(* IEC 61131-3 sources: Lua/ (part 2) *)

(* ---- ValveControl.st ---- *)
REGION 预处理
    #"FP-valve-Product"(CLK := #"Comm-Valve"."bnt-run");
    #"FP-valve-Manual"(CLK := #"Comm-Valve"."bnt-stop");
    #"Valve-Timer"[0](IN := #"Comm-Valve".busy,PT := #"Screen-Time"."PT-pretime-v");
    #"Valve-Timer"[1](IN := #"Comm-Valve"."in-timer".%X1,PT := #"Screen-Time"."PT-opentime");
    #"Valve-Timer"[2](IN := #"Comm-Valve"."in-timer".%X2,PT := #"Screen-Time"."PT-delaytime");
    #"Valve-Timer"[3](IN := #"Comm-Valve"."in-timer".%X3,PT := #"Screen-Time"."PT-looptime");
    //阀组生产模式
    IF "Debug".Unit_estop_state[2] THEN
        IF (#"FP-valve-Product".Q OR #"Comm-run".todo) AND NOT #"Comm-Valve".busy THEN
            #"Comm-Valve".todo := 1;
        END_IF;
        IF #"Comm-Valve".todo THEN
            #"Comm-Valve".busy := 1;
            #"Comm-Valve".step := 1;
            #"Comm-Valve".todo := 0;
        END_IF;
    ELSE
        #"Comm-Valve"."in-timer" := 0;
        #"Comm-Valve".todo := 0;
        #"Comm-Valve".busy := 0;
        #"Comm-Valve".step := 0;
    END_IF;
    //阀组手动模式
    IF "Debug".Unit_estop_state[2] THEN
        IF (#"FP-valve-Manual".Q OR #"Comm-stop".todo) THEN
            #"Comm-Valve"."in-timer" := 0;
            #"Comm-Valve".todo := 0;
            #"Comm-Valve".busy := 0;
            #"Comm-Valve".step := 0;
            "V5002-O" := 0;
            "V5003-O" := 0;
            "V5004-O" := 0;
            "V5101-O" := 0;
            "V5201-O" := 0;
        END_IF;
    END_IF;
END_REGION
REGION 冲洗阀组生产模式
    IF #"Comm-Valve".busy AND #"Valve-Timer"[0].Q THEN
        //step 1
        IF #"Comm-Valve".step = 1 THEN
            "V5201-O" := 1;
            #"Comm-Valve"."in-timer".%X1 := 1;
            IF #"Comm-Valve"."in-timer".%X1 AND #"Valve-Timer"[1].Q THEN
                "V5201-O" := 0;
                #"Comm-Valve"."in-timer".%X1 := 0;
                #"Comm-Valve"."in-timer".%X2 := 1;
                #"Comm-Valve".step := 2;
            END_IF;
        END_IF;
        //step 2
        IF #"Comm-Valve".step = 2 THEN
            IF #"Comm-Valve"."in-timer".%X2 AND #"Valve-Timer"[2].Q THEN
                "V5004-O" := 1;
                #"Comm-Valve"."in-timer".%X1 := 1;
                #"Comm-Valve"."in-timer".%X2 := 0;
            END_IF;
            IF #"Comm-Valve"."in-timer".%X1 AND #"Valve-Timer"[1].Q THEN
                "V5004-O" := 0;
                #"Comm-Valve"."in-timer".%X1 := 0;
                #"Comm-Valve"."in-timer".%X2 := 1;
                #"Comm-Valve".step := 3;
            END_IF;
        END_IF;
        //step 3
        IF #"Comm-Valve".step = 3 THEN
            IF #"Comm-Valve"."in-timer".%X2 AND #"Valve-Timer"[2].Q THEN
                "V5003-O" := 1;
                #"Comm-Valve"."in-timer".%X1 := 1;
                #"Comm-Valve"."in-timer".%X2 := 0;
            END_IF;
            IF #"Comm-Valve"."in-timer".%X1 AND #"Valve-Timer"[1].Q THEN
                "V5003-O" := 0;
                #"Comm-Valve"."in-timer".%X1 := 0;
                #"Comm-Valve"."in-timer".%X2 := 1;
                #"Comm-Valve".step := 4;
            END_IF;
        END_IF;
        //step 4
        IF #"Comm-Valve".step = 4 THEN
            IF #"Comm-Valve"."in-timer".%X2 AND #"Valve-Timer"[2].Q THEN
                "V5002-O" := 1;
                #"Comm-Valve"."in-timer".%X1 := 1;
                #"Comm-Valve"."in-timer".%X2 := 0;
            END_IF;
            IF #"Comm-Valve"."in-timer".%X1 AND #"Valve-Timer"[1].Q THEN
                "V5002-O" := 0;
                #"Comm-Valve"."in-timer".%X1 := 0;
                #"Comm-Valve"."in-timer".%X2 := 1;
                #"Comm-Valve".step := 5;
            END_IF;
        END_IF;
        //step 5
        IF #"Comm-Valve".step = 5 THEN
            IF #"Comm-Valve"."in-timer".%X2 AND #"Valve-Timer"[2].Q THEN
                "V5101-O" := 1;
                #"Comm-Valve"."in-timer".%X1 := 1;
                #"Comm-Valve"."in-timer".%X2 := 0;
            END_IF;
            IF #"Comm-Valve"."in-timer".%X1 AND #"Valve-Timer"[1].Q THEN
                "V5101-O" := 0;
                #"Comm-Valve"."in-timer".%X1 := 0;
                #"Comm-Valve"."in-timer".%X3 := 1;
            END_IF;
            IF #"Comm-Valve"."in-timer".%X3 AND #"Valve-Timer"[3].Q THEN
                #"Comm-Valve"."in-timer".%X3 := 0;
                #"Comm-Valve".step := 1;
            END_IF;
        END_IF;
    END_IF;
END_REGION

(* ---- ValveLoopControl_v1.0.st ---- *)
REGION 预处理
    #"FP-valve-Product"(CLK := #"Comm-Valve"."bnt-run");
    #"FP-valve-Manual"(CLK := #"Comm-Valve"."bnt-stop");
    #"Valve-Timer"[0](IN := #"Comm-Valve".busy,
                      PT := #"Screen-Time"."PT-pretime-v");
    #"Valve-Timer"[1](IN := #"Comm-Valve"."in-timer".%X1,
                      PT := #"Screen-Time"."PT-opentime");
    #"Valve-Timer"[2](IN := #"Comm-Valve"."in-timer".%X2,
                      PT := #"Screen-Time"."PT-delaytime");
    #"Valve-Timer"[3](IN := #"Comm-Valve"."in-timer".%X3,
                      PT := #"Screen-Time"."PT-looptime");
    //阀组生产模式
    IF "Debug".Unit_estop_state[2] THEN
        IF (#"FP-valve-Product".Q OR #"Comm-run".todo) AND NOT #"Comm-Valve".busy THEN
            #"Comm-Valve".todo := 1;
        END_IF;
        IF #"Comm-Valve".todo THEN
            #"Comm-Valve".busy := 1;
            #"Comm-Valve".step := 1;
            #"Comm-Valve".todo := 0;
        END_IF;
    ELSE
        #"Comm-Valve"."in-timer" := 0;
        #"Comm-Valve".todo := 0;
        #"Comm-Valve".busy := 0;
        #"Comm-Valve".step := 0;
    END_IF;
    //阀组手动模式
    IF "Debug".Unit_estop_state[2] THEN
        IF (#"FP-valve-Manual".Q OR #"Comm-stop".todo) THEN
            #"Comm-Valve"."in-timer" := 0;
            #"Comm-Valve".todo := 0;
            #"Comm-Valve".busy := 0;
            #"Comm-Valve".step := 0;
            "V5002-O" := 0;
            "V5003-O" := 0;
            "V5004-O" := 0;
            "V5101-O" := 0;
            "V5201-O" := 0;
        END_IF;
    END_IF;
END_REGION
REGION 冲洗阀组生产模式
    IF #"Comm-Valve".busy AND #"Valve-Timer"[0].Q THEN
        //step 1
        IF #"Comm-Valve".step = 1 THEN
            "V5201-O" := 1;
            #"Comm-Valve"."in-timer".%X1 := 1;
            IF #"Comm-Valve"."in-timer".%X1 AND #"Valve-Timer"[1].Q THEN
                "V5201-O" := 0;
                #"Comm-Valve"."in-timer".%X1 := 0;
                #"Comm-Valve"."in-timer".%X2 := 1;
                #"Comm-Valve".step := 2;
            END_IF;
        END_IF;
        //step 2
        IF #"Comm-Valve".step = 2 THEN
            IF #"Comm-Valve"."in-timer".%X2 AND #"Valve-Timer"[2].Q THEN
                "V5004-O" := 1;
                #"Comm-Valve"."in-timer".%X1 := 1;
                #"Comm-Valve"."in-timer".%X2 := 0;
            END_IF;
            IF #"Comm-Valve"."in-timer".%X1 AND #"Valve-Timer"[1].Q THEN
                "V5004-O" := 0;
                #"Comm-Valve"."in-timer".%X1 := 0;
                #"Comm-Valve"."in-timer".%X2 := 1;
                #"Comm-Valve".step := 3;
            END_IF;
        END_IF;
        //step 3
        IF #"Comm-Valve".step = 3 THEN
            IF #"Comm-Valve"."in-timer".%X2 AND #"Valve-Timer"[2].Q THEN
                "V5003-O" := 1;
                #"Comm-Valve"."in-timer".%X1 := 1;
                #"Comm-Valve"."in-timer".%X2 := 0;
            END_IF;
            IF #"Comm-Valve"."in-timer".%X1 AND #"Valve-Timer"[1].Q THEN
                "V5003-O" := 0;
                #"Comm-Valve"."in-timer".%X1 := 0;
                #"Comm-Valve"."in-timer".%X2 := 1;
                #"Comm-Valve".step := 4;
            END_IF;
        END_IF;
        //step 4
        IF #"Comm-Valve".step = 4 THEN
            IF #"Comm-Valve"."in-timer".%X2 AND #"Valve-Timer"[2].Q THEN
                "V5002-O" := 1;
                #"Comm-Valve"."in-timer".%X1 := 1;
                #"Comm-Valve"."in-timer".%X2 := 0;
            END_IF;
            IF #"Comm-Valve"."in-timer".%X1 AND #"Valve-Timer"[1].Q THEN
                "V5002-O" := 0;
                #"Comm-Valve"."in-timer".%X1 := 0;
                #"Comm-Valve"."in-timer".%X2 := 1;
                #"Comm-Valve".step := 5;
            END_IF;
        END_IF;
        //step 5
        IF #"Comm-Valve".step = 5 THEN
            IF #"Comm-Valve"."in-timer".%X2 AND #"Valve-Timer"[2].Q THEN
                "V5101-O" := 1;
                #"Comm-Valve"."in-timer".%X1 := 1;
                #"Comm-Valve"."in-timer".%X2 := 0;
            END_IF;
            IF #"Comm-Valve"."in-timer".%X1 AND #"Valve-Timer"[1].Q THEN
                "V5101-O" := 0;
                #"Comm-Valve"."in-timer".%X1 := 0;
                #"Comm-Valve"."in-timer".%X3 := 1;
            END_IF;
            IF #"Comm-Valve"."in-timer".%X3 AND #"Valve-Timer"[3].Q THEN
                #"Comm-Valve"."in-timer".%X3 := 0;
                #"Comm-Valve".step := 1;
            END_IF;
        END_IF;
    END_IF;
END_REGION

(* ---- Wash.st ---- *)
//自动放料回料控制
IF ("Databas".Xuanliu_V50XX_Tab = 1) THEN
    IF ("Databas".自动模式放料) THEN                   //放料控制

        "V5007-O" := 0;

        IF "Databas".放料通道选择 = 1 THEN
            "V5001-O" := TRUE;
            "V5002-O" := FALSE;

            //去4#反应罐
            IF "Databas".反应罐通道选择 = 1 THEN

                "V5004-O" := TRUE;
                "V5006-O" := TRUE;

                "V5003-O" := FALSE;
                "V5005-O" := FALSE;
            END_IF;

            //去5#反应罐
            IF "Databas".反应罐通道选择 = 2 THEN

                "V5004-O" := TRUE;
                "V5005-O" := TRUE;

                "V5003-O" := FALSE;
                "V5006-O" := FALSE;
            END_IF;

            //去6#反应罐
            IF "Databas".反应罐通道选择 = 3 THEN

                "V5003-O" := TRUE;

                "V5004-O" := FALSE;
                "V5005-O" := FALSE;
                "V5006-O" := FALSE;
            END_IF;
        END_IF;

        IF "Databas".放料通道选择 = 2 THEN
            "V5001-O" := FALSE;
            "V5002-O" := TRUE;
        END_IF;
    END_IF;

    IF ("Databas".自动模式回料) THEN                  //回料控制

        "V5007-O" := 1;
        "V5001-O" := FALSE;
        "V5002-O" := FALSE;
    END_IF;
END_IF;

//......2023-10-19 @smslule现场修改
IF "Databas".Xuanliu_V50XX_Tab = 0 THEN

    IF ("Databas".手动放料按钮) THEN
    //手动放料控制
        "V5007-O" := 0;
        IF "Databas".放料通道选择 = 1 THEN
            "V5001-O" := TRUE;
            "V5002-O" := FALSE;

            //去4#反应罐
            IF "Databas".反应罐通道选择 = 1 THEN

                "V5004-O" := TRUE;
                "V5006-O" := TRUE;

                "V5003-O" := FALSE;
                "V5005-O" := FALSE;

            END_IF;

            //去5#反应罐
            IF "Databas".反应罐通道选择 = 2 THEN

                "V5004-O" := TRUE;
                "V5005-O" := TRUE;

                "V5003-O" := FALSE;
                "V5006-O" := FALSE;

            END_IF;

            //去6#反应罐
            IF "Databas".反应罐通道选择 = 3 THEN

                "V5003-O" := TRUE;

                "V5004-O" := FALSE;
                "V5005-O" := FALSE;
                "V5006-O" := FALSE;

            END_IF;

        END_IF;

        IF "Databas".放料通道选择 = 2 THEN
            "V5001-O" := FALSE;
            "V5002-O" := TRUE;

        END_IF;

        "Databas".手动放料按钮 := FALSE;

    END_IF;

    IF ("Databas".手动回料按钮) THEN
    //手动回料控制
        "V5007-O" := 1;
        "V5001-O" := FALSE;
        "V5002-O" := FALSE;

        "Databas".手动回料按钮 := FALSE;

    END_IF;

    IF "Databas".手动淀粉乳阀 THEN

        "V5007-O" := 0;
        "V5001-O" := 0;
        "V5003-O" := 0;
        "V5004-O" := 0;
        "V5005-O" := 0;
        "V5006-O" := 0;
        "V5002-O" := 1;
        "Databas".手动淀粉乳阀 := FALSE;
    END_IF;

    IF "Databas".手动反应罐阀 THEN

        "V5007-O" := 0;
        "V5002-O" := 0;
        "V5001-O" := 1;
        "Databas".手动反应罐阀 := FALSE;
    END_IF;

    IF "Databas"."手动4#罐阀" THEN

        "V5007-O" := 0;
        "V5002-O" := 0;

        "V5003-O" := 0;
        "V5004-O" := 1;
        "V5005-O" := 0;
        "V5006-O" := 1;

        "V5001-O" := 1;
        "Databas"."手动4#罐阀" := FALSE;
    END_IF;

    IF "Databas"."手动5#罐阀" THEN

        "V5007-O" := 0;
        "V5002-O" := 0;

        "V5003-O" := 0;
        "V5004-O" := 1;
        "V5005-O" := 1;
        "V5006-O" := 0;

        "V5001-O" := 1;
        "Databas"."手动5#罐阀" := FALSE;
    END_IF;

    IF "Databas"."手动6#罐阀" THEN

        "V5007-O" := 0;
        "V5002-O" := 0;

        "V5003-O" := 1;
        "V5004-O" := 0;
        "V5005-O" := 0;
        "V5006-O" := 0;

        "V5001-O" := 1;
        "Databas"."手动6#罐阀" := FALSE;
    END_IF;

END_IF;

IF "V5002-O" OR "V5001-O" THEN
    "Databas".放料状态显示 := 1;

END_IF;

IF "V5002-O"=0 AND "V5001-O"=0 THEN
    "Databas".放料状态显示 := 2;

END_IF;

IF "Databas".反应罐方向按钮 THEN

    "Databas".放料通道选择 := 1;
    "Databas".反应罐方向按钮 := FALSE;
END_IF;

IF "Databas".淀粉乳罐方向按钮 THEN
        "Databas".反应罐通道选择 := 0;
        "Databas".放料通道选择 := 2;
        "Databas".淀粉乳罐方向按钮 := FALSE;
    END_IF;

//选择4#反应罐
    IF "Databas".反应罐方向1按钮 THEN

        "Databas".放料通道选择 := 1;
        "Databas".反应罐通道选择 := 1;
        "Databas".反应罐方向1按钮 := FALSE;
    END_IF;

//选择5#反应罐
    IF "Databas".反应罐方向2按钮 THEN
        "Databas".放料通道选择 := 1;
        "Databas".反应罐通道选择 := 2;
        "Databas".反应罐方向2按钮 := FALSE;
    END_IF;

//选择6#反应罐
    IF "Databas".反应罐方向3按钮 THEN
        "Databas".放料通道选择 := 1;
        "Databas".反应罐通道选择 := 3;
        "Databas".反应罐方向3按钮 := FALSE;
    END_IF;

IF (("Databas".Xuanliu_V50XX_Tab = 1) AND ("Databas".DIT5001_AI < "Databas".Xuanliu_DIT5001_L)) THEN
    "Databas".自动模式回料 := TRUE;
    "Databas".自动模式放料 := FALSE;
END_IF;

IF (("Databas".Xuanliu_V50XX_Tab = 1) AND ("Databas".DIT5001_AI > "Databas".Xuanliu_DIT5001_H)) THEN
    "Databas".自动模式放料 := TRUE;
    "Databas".自动模式回料 := FALSE;
END_IF;

(* ---- 放料回料控制.st ---- *)
//自动模式
IF "Debug".Unit_estop_state[3] AND #Valve.mode = 1 THEN
    IF "Global"."DIT6001-density" < #Retain."density-Low" THEN
        "V6003-O" := 1;
        "V6004-O" := 0;
    END_IF;
    IF "Global"."DIT6001-density" > #Retain."density-High" THEN
        "V6003-O" := 0;
        "V6004-O" := 1;
    END_IF;
END_IF;
//手动模式
IF "Debug".Unit_estop_state[3] AND #Valve.mode = 2 THEN
    IF #Valve."bnt-loop" THEN
        "V6003-O" := 1;
        "V6004-O" := 0;
    END_IF;
    IF #Valve."bnt-dump" THEN
        "V6003-O" := 0;
        "V6004-O" := 1;
    END_IF;
END_IF;
//急停模式下复位
IF NOT "Debug".Unit_estop_state[3] THEN
    "V6003-O" := 1;
    "V6004-O" := 0;
    #Valve.mode := 2;
END_IF;
//回料--放料状态判断
IF "V6003-O" AND NOT "V6004-O" THEN
    #Valve.state := 1;
END_IF;
IF NOT "V6003-O" AND "V6004-O" THEN
    #Valve.state := 2;
END_IF;
IF NOT "V6003-O" AND NOT "V6004-O" THEN
    #Valve.state := 0;
END_IF;
IF "V6003-O" AND "V6004-O" THEN
    #Valve.state := 3;
END_IF;

(* ---- 阀组控制.st ---- *)
REGION 预处理
    #"FP-valve-Product"(CLK := #"Comm-Valve"."bnt-run");
    #"FP-valve-Manual"(CLK := #"Comm-Valve"."bnt-stop");
    #"Valve-Timer"[0](IN := #"Comm-Valve".busy,PT := #"Screen-Time"."PT-pretime-v");
    #"Valve-Timer"[1](IN := #"Comm-Valve"."in-timer".%X1,PT := #"Screen-Time"."PT-opentime");
    #"Valve-Timer"[2](IN := #"Comm-Valve"."in-timer".%X2,PT := #"Screen-Time"."PT-delaytime");
    #"Valve-Timer"[3](IN := #"Comm-Valve"."in-timer".%X3,PT := #"Screen-Time"."PT-looptime");
    //阀组生产模式
    IF "Debug".Unit_estop_state[2] THEN
        IF (#"FP-valve-Product".Q OR #"Comm-run".todo) AND NOT #"Comm-Valve".busy THEN
            #"Comm-Valve".todo := 1;
        END_IF;
        IF #"Comm-Valve".todo THEN
            #"Comm-Valve".busy := 1;
            #"Comm-Valve".step := 1;
            #"Comm-Valve".todo := 0;
        END_IF;
    ELSE
        #"Comm-Valve"."in-timer" := 0;
        #"Comm-Valve".todo := 0;
        #"Comm-Valve".busy := 0;
        #"Comm-Valve".step := 0;
    END_IF;
    //阀组手动模式
    IF "Debug".Unit_estop_state[2] THEN
        IF (#"FP-valve-Manual".Q OR #"Comm-stop".todo) THEN
            #"Comm-Valve"."in-timer" := 0;
            #"Comm-Valve".todo := 0;
            #"Comm-Valve".busy := 0;
            #"Comm-Valve".step := 0;
            "V5002-O" := 0;
            "V5003-O" := 0;
            "V5004-O" := 0;
            "V5101-O" := 0;
            "V5201-O" := 0;
        END_IF;
    END_IF;
END_REGION
REGION 冲洗阀组生产模式
    IF #"Comm-Valve".busy AND #"Valve-Timer"[0].Q THEN
        //step 1
        IF #"Comm-Valve".step = 1 THEN
            "V5201-O" := 1;
            #"Comm-Valve"."in-timer".%X1 := 1;
            IF #"Comm-Valve"."in-timer".%X1 AND #"Valve-Timer"[1].Q THEN
                "V5201-O" := 0;
                #"Comm-Valve"."in-timer".%X1 := 0;
                #"Comm-Valve"."in-timer".%X2 := 1;
                #"Comm-Valve".step := 2;
            END_IF;
        END_IF;
        //step 2
        IF #"Comm-Valve".step = 2 THEN
            IF #"Comm-Valve"."in-timer".%X2 AND #"Valve-Timer"[2].Q THEN
                "V5004-O" := 1;
                #"Comm-Valve"."in-timer".%X1 := 1;
                #"Comm-Valve"."in-timer".%X2 := 0;
            END_IF;
            IF #"Comm-Valve"."in-timer".%X1 AND #"Valve-Timer"[1].Q THEN
                "V5004-O" := 0;
                #"Comm-Valve"."in-timer".%X1 := 0;
                #"Comm-Valve"."in-timer".%X2 := 1;
                #"Comm-Valve".step := 3;
            END_IF;
        END_IF;
        //step 3
        IF #"Comm-Valve".step = 3 THEN
            IF #"Comm-Valve"."in-timer".%X2 AND #"Valve-Timer"[2].Q THEN
                "V5003-O" := 1;
                #"Comm-Valve"."in-timer".%X1 := 1;
                #"Comm-Valve"."in-timer".%X2 := 0;
            END_IF;
            IF #"Comm-Valve"."in-timer".%X1 AND #"Valve-Timer"[1].Q THEN
                "V5003-O" := 0;
                #"Comm-Valve"."in-timer".%X1 := 0;
                #"Comm-Valve"."in-timer".%X2 := 1;
                #"Comm-Valve".step := 4;
            END_IF;
        END_IF;
        //step 4
        IF #"Comm-Valve".step = 4 THEN
            IF #"Comm-Valve"."in-timer".%X2 AND #"Valve-Timer"[2].Q THEN
                "V5002-O" := 1;
                #"Comm-Valve"."in-timer".%X1 := 1;
                #"Comm-Valve"."in-timer".%X2 := 0;
            END_IF;
            IF #"Comm-Valve"."in-timer".%X1 AND #"Valve-Timer"[1].Q THEN
                "V5002-O" := 0;
                #"Comm-Valve"."in-timer".%X1 := 0;
                #"Comm-Valve"."in-timer".%X2 := 1;
                #"Comm-Valve".step := 5;
            END_IF;
        END_IF;
        //step 5
        IF #"Comm-Valve".step = 5 THEN
            IF #"Comm-Valve"."in-timer".%X2 AND #"Valve-Timer"[2].Q THEN
                "V5101-O" := 1;
                #"Comm-Valve"."in-timer".%X1 := 1;
                #"Comm-Valve"."in-timer".%X2 := 0;
            END_IF;
            IF #"Comm-Valve"."in-timer".%X1 AND #"Valve-Timer"[1].Q THEN
                "V5101-O" := 0;
                #"Comm-Valve"."in-timer".%X1 := 0;
                #"Comm-Valve"."in-timer".%X3 := 1;
            END_IF;
            IF #"Comm-Valve"."in-timer".%X3 AND #"Valve-Timer"[3].Q THEN
                #"Comm-Valve"."in-timer".%X3 := 0;
                #"Comm-Valve".step := 1;
            END_IF;
        END_IF;
    END_IF;
END_REGION

REGION V4001预处理
    #"Desand-Timer-1"[0](IN := #"Comm-desand-1".busy,
                         PT := #"Desand-Time"."PT-pretime");
    #"Desand-Timer-1"[1](IN := #"Comm-desand-1"."in-timer".%X1,
                         PT := #"Desand-Time"."PT-opentime");
    #"Desand-Timer-1"[2](IN := #"Comm-desand-1"."in-timer".%X2,
                         PT := #"Desand-Time"."PT-looptime");
    //生产模式
    IF "Debug".Unit_estop_state[2] THEN
        IF #"Comm-desand-1"."bnt-run" AND NOT #"Comm-desand-1".busy THEN
            #"Comm-desand-1".todo := 1;
        END_IF;
        IF #"Comm-desand-1".todo THEN
            #"Comm-desand-1".busy := 1;
            #"Comm-desand-1".step := 1;
            #"Comm-desand-1".todo := 0;
        END_IF;
    ELSE
        #"Comm-desand-1"."in-timer" := 0;
        #"Comm-desand-1".todo := 0;
        #"Comm-desand-1".busy := 0;
        #"Comm-desand-1".step := 0;
    END_IF;
    //手动模式
    IF "Debug".Unit_estop_state[2] THEN
        IF #"Comm-desand-1"."bnt-stop" THEN
            #"Comm-desand-1"."in-timer" := 0;
            #"Comm-desand-1".todo := 0;
            #"Comm-desand-1".busy := 0;
            #"Comm-desand-1".step := 0;
            "V4001-O" := 0;
        END_IF;
    END_IF;
END_REGION
REGION V4001生产模式
    IF #"Comm-desand-1".busy AND #"Desand-Timer-1"[0].Q THEN
        //step 1
        IF #"Comm-desand-1".step = 1 THEN
            "V4001-O" := 1;
            #"Comm-desand-1"."in-timer".%X1 := 1;
            IF #"Comm-desand-1"."in-timer".%X1 AND #"Desand-Timer-1"[1].Q THEN
                "V4001-O" := 0;
                #"Comm-desand-1"."in-timer".%X1 := 0;
                #"Comm-desand-1"."in-timer".%X2 := 1;
                #"Comm-desand-1".step := 2;
            END_IF;
        END_IF;
        //step 2
        IF #"Comm-desand-1".step = 2 THEN
            IF #"Comm-desand-1"."in-timer".%X2 AND #"Desand-Timer-1"[2].Q THEN
                #"Comm-desand-1"."in-timer".%X2 := 0;
                #"Comm-desand-1".step := 1;
            END_IF;
        END_IF;
    END_IF;
END_REGION
REGION V6005预处理
    #"Desand-Timer-2"[0](IN := #"Comm-desand-2".busy,
                         PT := #"Desand-Time"."PT-pretime");
    #"Desand-Timer-2"[1](IN := #"Comm-desand-2"."in-timer".%X1,
                         PT := #"Desand-Time"."PT-opentime");
    #"Desand-Timer-2"[2](IN := #"Comm-desand-2"."in-timer".%X2,
                         PT := #"Desand-Time"."PT-looptime");
    //生产模式
    IF "Debug".Unit_estop_state[2] THEN
        IF #"Comm-desand-2"."bnt-run" AND NOT #"Comm-desand-2".busy THEN
            #"Comm-desand-2".todo := 1;
        END_IF;
        IF #"Comm-desand-2".todo THEN
            #"Comm-desand-2".busy := 1;
            #"Comm-desand-2".step := 1;
            #"Comm-desand-2".todo := 0;
        END_IF;
    ELSE
        #"Comm-desand-2"."in-timer" := 0;
        #"Comm-desand-2".todo := 0;
        #"Comm-desand-2".busy := 0;
        #"Comm-desand-2".step := 0;
    END_IF;
    //手动模式
    IF "Debug".Unit_estop_state[2] THEN
        IF #"Comm-desand-2"."bnt-stop" THEN
            #"Comm-desand-2"."in-timer" := 0;
            #"Comm-desand-2".todo := 0;
            #"Comm-desand-2".busy := 0;
            #"Comm-desand-2".step := 0;
            "V6005-O" := 0;
        END_IF;
    END_IF;
END_REGION
REGION V6005生产模式
    IF #"Comm-desand-2".busy AND #"Desand-Timer-2"[0].Q THEN
        //step 1
        IF #"Comm-desand-2".step = 1 THEN
            "V6005-O" := 1;
            #"Comm-desand-2"."in-timer".%X1 := 1;
            IF #"Comm-desand-2"."in-timer".%X1 AND #"Desand-Timer-2"[1].Q THEN
                "V6005-O" := 0;
                #"Comm-desand-2"."in-timer".%X1 := 0;
                #"Comm-desand-2"."in-timer".%X2 := 1;
                #"Comm-desand-2".step := 2;
            END_IF;
        END_IF;
        //step 2
        IF #"Comm-desand-2".step = 2 THEN
            IF #"Comm-desand-2"."in-timer".%X2 AND #"Desand-Timer-2"[2].Q THEN
                #"Comm-desand-2"."in-timer".%X2 := 0;
                #"Comm-desand-2".step := 1;
            END_IF;
        END_IF;
    END_IF;
END_REGION

(* ---- 顺序启动_0521.st ---- *)
/* *
**计时器
 */
#Timer_M5000_run[0](IN := #Common_M_1_run.in_time.%X0, PT := #Retain_M5000_run.preTime);
#Timer_M5000_run[1](IN := #Common_M_1_run.in_time.%X1, PT := #Retain_M5000_run.openTime_1);
/* *
**预处理
 */
IF "Global".Emergency.Extraction_1 AND #Common_M_1_run.bnt_run AND NOT #Common_M_1_run.busy THEN
    #Common_M_1_run.state := 1;
    #Common_M_1_run.STEP := 1;
    #Common_M_1_run.in_time := 0;
    #Common_M_1_run.todo := FALSE;
    #Common_M_1_run.in_time.%X0 := TRUE;
END_IF;
IF #Common_M_1_run.in_time.%X0 AND #Timer_M5000_run[0].Q THEN
    #Common_M_1_run.bnt_run := FALSE;
    #Common_M_1_run.busy := TRUE;
ELSE
    #Common_M_1_run.busy := FALSE;
END_IF;
//急停时
IF NOT "Global".Emergency.Extraction_1 THEN
    #Common_M_1_run.state := 0;
    #Common_M_1_run.STEP := 0;
    #Common_M_1_run.in_time := 0;
    #Common_M_1_run.bnt_run := FALSE;
END_IF;
//手动时
IF "Global".Emergency.Extraction_1 AND #Common_M_1_run.manual_enable THEN
    #Common_M_1_run.state := 2;
    #Common_M_1_run.STEP := 0;
    #Common_M_1_run.in_time := 0;
    #Common_M_1_run.bnt_run := FALSE;
END_IF;
//停止时
IF "Global".Emergency.Extraction_1 AND #Common_M_1_run.bnt_stop THEN
    #Common_M_1_run.STEP := 0;
    #Common_M_1_run.in_time := 0;
    #Common_M_1_run.bnt_run := FALSE;
END_IF;
/* *
**运行时
 */
 IF #Common_M_1_run.busy AND #Common_M_1_run.state = 1 THEN
    //step1
    IF #Common_M_1_run.step = 1 THEN
        IF NOT "M5203-DO" THEN
            "M5203-DO" := TRUE;
            #Common_M_1_run.step := 2;
            RETURN;
        END_IF;
        IF "M5203-DO" THEN
            #Common_M_1_run.todo := TRUE;
            #Common_M_1_run.step := 2;
        END_IF;
    END_IF;
    //step2
    IF #Common_M_1_run.step = 2 THEN
        IF NOT "M5103-DO" THEN
            IF #Common_M_1_run.todo THEN
                "M5103-DO" := TRUE;
                #Common_M_1_run.todo := FALSE;
                #Common_M_1_run.step := 3;
                RETURN;
            END_IF;
            #Common_M_1_run.in_time.%X1 := TRUE;
            IF #Common_M_1_run.in_time.%X1 AND #Timer_M5000_run[1].Q THEN
                "M5103-DO" := TRUE;
                #Common_M_1_run.in_time.%X1 := FALSE;
                #Common_M_1_run.step := 3;
                RETURN;
            END_IF;
        END_IF;
        IF "M5103-DO" THEN
            #Common_M_1_run.step := 3;
        END_IF;
    END_IF;
    //step3
    IF #Common_M_1_run.step = 3 THEN
        IF NOT "M5202-DO" THEN
            IF #Common_M_1_run.todo THEN
                "M5202-DO" := TRUE;
                #Common_M_1_run.todo := FALSE;
                #Common_M_1_run.step := 4;
                RETURN;
            END_IF;
            #Common_M_1_run.in_time.%X1 := TRUE;
            IF #Common_M_1_run.in_time.%X1 AND #Timer_M5000_run[1].Q THEN
                "M5202-DO" := TRUE;
                #Common_M_1_run.in_time.%X1 := FALSE;
                #Common_M_1_run.step := 4;
                RETURN;
            END_IF;
        END_IF;
        IF "M5202-DO" THEN
            #Common_M_1_run.step := 4;
        END_IF;
    END_IF;
    //step4
    IF #Common_M_1_run.step = 4 THEN
        IF NOT "M5102-DO" THEN
            IF #Common_M_1_run.todo THEN
                "M5102-DO" := TRUE;
                #Common_M_1_run.todo := FALSE;
                #Common_M_1_run.step := 5;
                RETURN;
            END_IF;
            #Common_M_1_run.in_time.%X1 := TRUE;
            IF #Common_M_1_run.in_time.%X1 AND #Timer_M5000_run[1].Q THEN
                "M5102-DO" := TRUE;
                #Common_M_1_run.in_time.%X1 := FALSE;
                #Common_M_1_run.step := 5;
                RETURN;
            END_IF;
        END_IF;
        IF "M5102-DO" THEN
            #Common_M_1_run.step := 5;
        END_IF;
    END_IF;
    //step5
    IF #Common_M_1_run.step = 5 THEN
        IF NOT "M5401-DO" THEN
            IF #Common_M_1_run.todo THEN
                "M5401-DO" := TRUE;
                #Common_M_1_run.todo := FALSE;
                #Common_M_1_run.step := 6;
                RETURN;
            END_IF;
            #Common_M_1_run.in_time.%X1 := TRUE;
            IF #Common_M_1_run.in_time.%X1 AND #Timer_M5000_run[1].Q THEN
                "M5401-DO" := TRUE;
                #Common_M_1_run.in_time.%X1 := FALSE;
                #Common_M_1_run.step := 6;
                RETURN;
            END_IF;
        END_IF;
        IF "M5401-DO" THEN
            #Common_M_1_run.step := 6;
        END_IF;
    END_IF;
    //step6
    IF #Common_M_1_run.step = 6 THEN
        IF NOT "M5301-DO" THEN
            IF #Common_M_1_run.todo THEN
                "M5301-DO" := TRUE;
                #Common_M_1_run.todo := FALSE;
                #Common_M_1_run.step := 7;
                RETURN;
            END_IF;
            #Common_M_1_run.in_time.%X1 := TRUE;
            IF #Common_M_1_run.in_time.%X1 AND #Timer_M5000_run[1].Q THEN
                "M5301-DO" := TRUE;
                #Common_M_1_run.in_time.%X1 := FALSE;
                #Common_M_1_run.step := 7;
                RETURN;
            END_IF;
        END_IF;
        IF "M5301-DO" THEN
            #Common_M_1_run.step := 7;
        END_IF;
    END_IF;
    //step7
    IF #Common_M_1_run.step = 7 THEN
        IF NOT "M5201-DO" THEN
            IF #Common_M_1_run.todo THEN
                "M5201-DO" := TRUE;
                #Common_M_1_run.todo := FALSE;
                #Common_M_1_run.step := 8;
                RETURN;
            END_IF;
            #Common_M_1_run.in_time.%X1 := TRUE;
            IF #Common_M_1_run.in_time.%X1 AND #Timer_M5000_run[1].Q THEN
                "M5201-DO" := TRUE;
                #Common_M_1_run.in_time.%X1 := FALSE;
                #Common_M_1_run.step := 8;
                RETURN;
            END_IF;
        END_IF;
        IF "M5201-DO" THEN
            #Common_M_1_run.step := 8;
        END_IF;
    END_IF;
    //step8
    IF #Common_M_1_run.step = 8 THEN
        IF NOT "M5101-DO" THEN
            IF #Common_M_1_run.todo THEN
                "M5101-DO" := TRUE;
                #Common_M_1_run.todo := FALSE;
                #Common_M_1_run.step := 9;
                RETURN;
            END_IF;
            #Common_M_1_run.in_time.%X1 := TRUE;
            IF #Common_M_1_run.in_time.%X1 AND #Timer_M5000_run[1].Q THEN
                "M5101-DO" := TRUE;
                #Common_M_1_run.in_time.%X1 := FALSE;
                #Common_M_1_run.step := 9;
                RETURN;
            END_IF;
        END_IF;
        IF "M5101-DO" THEN
            #Common_M_1_run.step := 9;
        END_IF;
    END_IF;
    //step9
    IF #Common_M_1_run.step = 9 THEN
        IF NOT "P5005-DO" THEN
            IF #Common_M_1_run.todo THEN
                "P5005-DO" := TRUE;
                #Common_M_1_run.todo := FALSE;
                #Common_M_1_run.step := 10;
                RETURN;
            END_IF;
            #Common_M_1_run.in_time.%X1 := TRUE;
            IF #Common_M_1_run.in_time.%X1 AND #Timer_M5000_run[1].Q THEN
                "P5005-DO" := TRUE;
                #Common_M_1_run.in_time.%X1 := FALSE;
                #Common_M_1_run.step := 10;
                RETURN;
            END_IF;
        END_IF;
        IF "P5005-DO" THEN
            #Common_M_1_run.step := 10;
        END_IF;
    END_IF;
    //step10
    IF #Common_M_1_run.step = 10 THEN
        IF NOT "P5003-DO" THEN
            IF #Common_M_1_run.todo THEN
                "P5003-DO" := TRUE;
                #Common_M_1_run.todo := FALSE;
                #Common_M_1_run.step := 11;
                RETURN;
            END_IF;
            #Common_M_1_run.in_time.%X1 := TRUE;
            IF #Common_M_1_run.in_time.%X1 AND #Timer_M5000_run[1].Q THEN
                "P5003-DO" := TRUE;
                #Common_M_1_run.in_time.%X1 := FALSE;
                #Common_M_1_run.step := 11;
                RETURN;
            END_IF;
        END_IF;
        IF "P5003-DO" THEN
            #Common_M_1_run.step := 11;
        END_IF;
    END_IF;
    //step11
    IF #Common_M_1_run.step = 11 THEN
        IF NOT "P5201-DO" THEN
            IF #Common_M_1_run.todo THEN
                "P5201-DO" := TRUE;
                #Common_M_1_run.todo := FALSE;
                #Common_M_1_run.step := 12;
                RETURN;
            END_IF;
            #Common_M_1_run.in_time.%X1 := TRUE;
            IF #Common_M_1_run.in_time.%X1 AND #Timer_M5000_run[1].Q THEN
                "P5201-DO" := TRUE;
                #Common_M_1_run.in_time.%X1 := FALSE;
                #Common_M_1_run.step := 12;
                RETURN;
            END_IF;
        END_IF;
        IF "P5201-DO" THEN
            #Common_M_1_run.step := 12;
        END_IF;
    END_IF;
    //step12
    IF #Common_M_1_run.step = 12 THEN
        IF NOT "P5101-DO" THEN
            IF #Common_M_1_run.todo THEN
                "P5101-DO" := TRUE;
                #Common_M_1_run.todo := FALSE;
                #Common_M_1_run.step := 13;
                RETURN;
            END_IF;
            #Common_M_1_run.in_time.%X1 := TRUE;
            IF #Common_M_1_run.in_time.%X1 AND #Timer_M5000_run[1].Q THEN
                "P5101-DO" := TRUE;
                #Common_M_1_run.in_time.%X1 := FALSE;
                #Common_M_1_run.step := 13;
                RETURN;
            END_IF;
        END_IF;
        IF "P5101-DO" THEN
            #Common_M_1_run.step := 13;
        END_IF;
    END_IF;
    //step13
    IF #Common_M_1_run.step = 13 THEN
        IF NOT "P5206-DO" THEN
            IF #Common_M_1_run.todo THEN
                "P5206-DO" := TRUE;
                #Common_M_1_run.todo := FALSE;
                #Common_M_1_run.step := 14;
                RETURN;
            END_IF;
            #Common_M_1_run.in_time.%X1 := TRUE;
            IF #Common_M_1_run.in_time.%X1 AND #Timer_M5000_run[1].Q THEN
                "P5206-DO" := TRUE;
                #Common_M_1_run.in_time.%X1 := FALSE;
                #Common_M_1_run.step := 14;
                RETURN;
            END_IF;
        END_IF;
        IF "P5206-DO" THEN
            #Common_M_1_run.step := 14;
        END_IF;
    END_IF;
    //step14
    IF #Common_M_1_run.step = 14 THEN
        IF NOT "P5106-DO" THEN
            IF #Common_M_1_run.todo THEN
                "P5106-DO" := TRUE;
                #Common_M_1_run.todo := FALSE;
                #Common_M_1_run.step := 15;
                RETURN;
            END_IF;
            #Common_M_1_run.in_time.%X1 := TRUE;
            IF #Common_M_1_run.in_time.%X1 AND #Timer_M5000_run[1].Q THEN
                "P5106-DO" := TRUE;
                #Common_M_1_run.in_time.%X1 := FALSE;
                #Common_M_1_run.step := 15;
                RETURN;
            END_IF;
        END_IF;
        IF "P5106-DO" THEN
            #Common_M_1_run.step := 15;
        END_IF;
    END_IF;
    //step15
    IF #Common_M_1_run.step = 15 THEN
        IF NOT "P5204-DO" THEN
            IF #Common_M_1_run.todo THEN
                "P5204-DO" := TRUE;
                #Common_M_1_run.todo := FALSE;
                #Common_M_1_run.step := 16;
                RETURN;
            END_IF;
            #Common_M_1_run.in_time.%X1 := TRUE;
            IF #Common_M_1_run.in_time.%X1 AND #Timer_M5000_run[1].Q THEN
                "P5204-DO" := TRUE;
                #Common_M_1_run.in_time.%X1 := FALSE;
                #Common_M_1_run.step := 16;
                RETURN;
            END_IF;
        END_IF;
        IF "P5204-DO" THEN
            #Common_M_1_run.step := 16;
        END_IF;
    END_IF;
    //step16
    IF #Common_M_1_run.step = 16 THEN
        IF NOT "P5104-DO" THEN
            IF #Common_M_1_run.todo THEN
                "P5104-DO" := TRUE;
                #Common_M_1_run.todo := FALSE;
                #Common_M_1_run.step := 17;
                RETURN;
            END_IF;
            #Common_M_1_run.in_time.%X1 := TRUE;
            IF #Common_M_1_run.in_time.%X1 AND #Timer_M5000_run[1].Q THEN
                "P5104-DO" := TRUE;
                #Common_M_1_run.in_time.%X1 := FALSE;
                #Common_M_1_run.step := 17;
                RETURN;
            END_IF;
        END_IF;
        IF "P5104-DO" THEN
            #Common_M_1_run.step := 17;
        END_IF;
    END_IF;
    //step17
    IF #Common_M_1_run.step = 17 THEN
        IF NOT "P5402-DO" THEN
            IF #Common_M_1_run.todo THEN
                "P5402-DO" := TRUE;
                #Common_M_1_run.todo := FALSE;
                #Common_M_1_run.step := 18;
                RETURN;
            END_IF;
            #Common_M_1_run.in_time.%X1 := TRUE;
            IF #Common_M_1_run.in_time.%X1 AND #Timer_M5000_run[1].Q THEN
                "P5402-DO" := TRUE;
                #Common_M_1_run.in_time.%X1 := FALSE;
                #Common_M_1_run.step := 18;
                RETURN;
            END_IF;
        END_IF;
        IF "P5402-DO" THEN
            #Common_M_1_run.step := 18;
        END_IF;
    END_IF;
    //step18
    IF #Common_M_1_run.step = 18 THEN
        IF NOT "P5302-DO" THEN
            IF #Common_M_1_run.todo THEN
                "P5302-DO" := TRUE;
                #Common_M_1_run.todo := FALSE;
                #Common_M_1_run.step := 19;
                RETURN;
            END_IF;
            #Common_M_1_run.in_time.%X1 := TRUE;
            IF #Common_M_1_run.in_time.%X1 AND #Timer_M5000_run[1].Q THEN
                "P5302-DO" := TRUE;
                #Common_M_1_run.in_time.%X1 := FALSE;
                #Common_M_1_run.step := 19;
                RETURN;
            END_IF;
        END_IF;
        IF "P5302-DO" THEN
            #Common_M_1_run.step := 19;
        END_IF;
    END_IF;
    //step19
    IF #Common_M_1_run.step = 19 THEN
        IF NOT "P5202-DO" THEN
            IF #Common_M_1_run.todo THEN
                "P5202-DO" := TRUE;
                #Common_M_1_run.todo := FALSE;
                #Common_M_1_run.step := 20;
                RETURN;
            END_IF;
            #Common_M_1_run.in_time.%X1 := TRUE;
            IF #Common_M_1_run.in_time.%X1 AND #Timer_M5000_run[1].Q THEN
                "P5202-DO" := TRUE;
                #Common_M_1_run.in_time.%X1 := FALSE;
                #Common_M_1_run.step := 20;
                RETURN;
            END_IF;
        END_IF;
        IF "P5202-DO" THEN
            #Common_M_1_run.step := 20;
        END_IF;
    END_IF;
    //step20
    IF #Common_M_1_run.step = 20 THEN
        IF NOT "P5102-DO" THEN
            IF #Common_M_1_run.todo THEN
                "P5102-DO" := TRUE;
                #Common_M_1_run.todo := FALSE;
                #Common_M_1_run.in_time := 0;
                #Common_M_1_run.step := 100;
                RETURN;
            END_IF;
            #Common_M_1_run.in_time.%X1 := TRUE;
            IF #Common_M_1_run.in_time.%X1 AND #Timer_M5000_run[1].Q THEN
                "P5102-DO" := TRUE;
                #Common_M_1_run.in_time := 0;
                #Common_M_1_run.step := 100;
                RETURN;
            END_IF;
        END_IF;
        IF "P5102-DO" THEN
            #Common_M_1_run.in_time := 0;
            #Common_M_1_run.step := 100;
        END_IF;
    END_IF;
END_IF;
